{attribute addProperty BoxType "AX8108-0000-0100-0100"}
{attribute addProperty Id "Ch_A_AxisMain_InputsCh_A_AxisMain_Inputs_70FF8C34648Ch_A_AxisMain_OutputsCh_A_AxisMain_Outputs_1B3A309C162Ch_A_Interpolator_OutputsCh_A_Interpolator_Outputs_70719997648Ch_A_PositionControl_InputsCh_A_PositionControl_Inputs_57B958FE324"}
{attribute addProperty CRC "899470490"}
{attribute addProperty SizeInBites "176"}
{attribute addProperty SizeInBytes "22"}
TYPE Ch_A_359CD49A :
STRUCT
	{attribute addProperty Name "Ch_A_AxisMain_Inputs"}
	Ch_A_AxisMain_Inputs  : Ch_A_AxisMain_Inputs_70FF8C34;
	{attribute addProperty Name "Ch_A_AxisMain_Outputs"}
	Ch_A_AxisMain_Outputs  : Ch_A_AxisMain_Outputs_1B3A309C;
	{attribute addProperty Name "Ch_A_Interpolator_Outputs"}
	Ch_A_Interpolator_Outputs  : Ch_A_Interpolator_Outputs_70719997;
	{attribute addProperty Name "Ch_A_PositionControl_Inputs"}
	Ch_A_PositionControl_Inputs  : Ch_A_PositionControl_Inputs_57B958FE;
END_STRUCT
END_TYPE

(* stored: Version 1.2.0.0, ProductVersion 3.1.4024.9
   DUT Ch_A_359CD49A: Id {d03c1a30-74b2-4de3-8974-e01bea8c40ea} *)
